(* CODESYS project MID_RunTime_Demo.project

Project tree, tasks and I/O mapping:
  Device : Changsha Xiangji-ARM Cortex A9(xilinx zynq7000)-linux, Changsha Xiangji Hiden Technology Co.Ltd, version 3.5.10.20
    application Application
      libraries: Standard, * (System); SysFile, * (System); SysTypes2 Interfaces, * (System)
      task MainTask (cyclic, interval 4 ms, priority 1) calls PLC_PRG
      task VISU_TASK (cyclic, interval 100 ms, priority 31) calls VisuElems.Visu_Prg
      program PLC_PRG [ST]
      function fn_set_Run_min [ST]
      function read_run_min [ST]
      visualisation RunTime_Visua
      global variables GVL
    SoftMotion General Axis Pool
  text list GlobalTextList
*)

// Device/Application/GVL
{attribute 'qualified_only'}
{attribute 'qualified_only'}


VAR_GLOBAL


	read_runmin:BOOL;
	boot_flag:BOOL;

END_VAR

// Device/Application/PLC_PRG
PROGRAM PLC_PRG
VAR
	Work_min:INT;
	Work_mins:STRING;
	Work_hour:REAL;
	ton1:TON;
	ton2:TON;
	
	new_Run_min:STRING;
	Run_min:STRING;
END_VAR

IF  gvl.boot_flag=FALSE THEN           //上电读一次小时计
   read_run_min(ADR(Work_mins));  //读小时计
   Work_min:=STRING_TO_INT(Work_mins);
   Work_hour:=ANY_TO_REAL(Work_min)/60;
    gvl.boot_flag:=TRUE;
END_IF



//更新小时计
	TON1(IN:=TRUE,PT:=T#60S);
		IF TON1.Q=TRUE THEN
				Work_min:=Work_min+1;		//每分钟加1
				new_Run_min:=INT_TO_STRING(Work_min);
                IF fn_set_Run_min(ADR(new_Run_min), len(new_Run_min)) THEN  //每分钟更新小时计后写入文件
	               Run_min := new_Run_min;
                END_IF				
				
			  TON1(IN:=FALSE,PT:=T#60S);
		END_IF
//读小时计（每6分钟即0.1h读一次）
	TON2(IN:=TRUE,PT:=T#360S);
		IF TON2.Q=TRUE THEN
	          read_run_min(ADR(Work_mins));  //读小时计
              Work_min:=STRING_TO_INT(Work_mins);
              Work_hour:=ANY_TO_REAL(Work_min)/60;	
			  TON2(IN:=FALSE,PT:=T#360S);
		END_IF

END_PROGRAM

// Device/Application/read_run_min
FUNCTION read_run_min : LINT
VAR_INPUT
	runmin: POINTER TO LINT;
END_VAR
VAR
	hFile: RTS_IEC_HANDLE;
	udiOpenError: RTS_IEC_RESULT;
	udiReadError: RTS_IEC_RESULT;
	i :INT;
	iTemp: UDINT;
	udiPos: UDINT;
	str_size: __XWORD;
	udiByteRead: LWORD;

	len_of_line: INT;
	len_of_number :INT;
	magicNumber:REAL;
	check_sum:REAL:= 0;
	temp_num:REAL;
END_VAR

gvl.read_runmin := FALSE;

//检测文件是否存在
hFile := sysfileopen(szFile := '/userapp/r_mins.txt', am := sysfile.AM_READ, pResult:= ADR(udiOpenError));
IF hFile = RTS_INVALID_HANDLE	THEN  //文件不存在
	RETURN;
END_IF
//文件存在，开始读取内容
udiPos := SysFileSetPos(hFile:=hFile, ulOffset := 0);
udiByteRead := sysfile.SysFileRead(hfile := hFile,pbyBuffer := runmin, ulSize := 32, pResult := ADR(udiReadError));
IF udiByteRead < 4 THEN  //读取失败
	sysfile.SysFileClose(hFile := hFile);
	RETURN;
END_IF

gvl.read_runmin := TRUE;

END_FUNCTION

// Device/Application/fn_set_Run_min
FUNCTION fn_set_Run_min : BOOL
VAR_INPUT
	Run_min: POINTER TO STRING;
	len:DINT;
END_VAR
VAR
	hFile: RTS_IEC_HANDLE;
	udiOpenError: RTS_IEC_RESULT;
	udiReadError: RTS_IEC_RESULT;
	udiWriteError: RTS_IEC_RESULT;
	i :INT;
	iTemp: UDINT;
	udiPos: UDINT;
	str_size: __XWORD;
	udiByteRead: UDINT;

	len_of_line: INT;
	len_of_number :INT;
	magicNumber:REAL;
	check_sum:REAL:= 0;
	temp_num:REAL;
	udiByteWrite: LWORD;
END_VAR


fn_set_Run_min := FALSE;

hFile := sysfileopen(szFile := '/userapp/r_mins.txt', am := sysfile.AM_WRITE, pResult := ADR(udiOpenError));
IF hFile = RTS_INVALID_HANDLE THEN //创建文件失败
	RETURN;
END_IF

udiPos := SysFileSetPos(hFile:=hFile, ulOffset:=0);	
udiByteWrite := sysfile.SysFileWrite(hFile := hFile,pbyBuffer := Run_min,ulSize := ANY_TO_DWORD(len), pResult := ADR(udiWriteError));
IF udiByteWrite = 0 THEN
	RETURN;
END_IF

fn_set_Run_min := TRUE;
RETURN;

END_FUNCTION

// Device/Application/RunTime_Visua
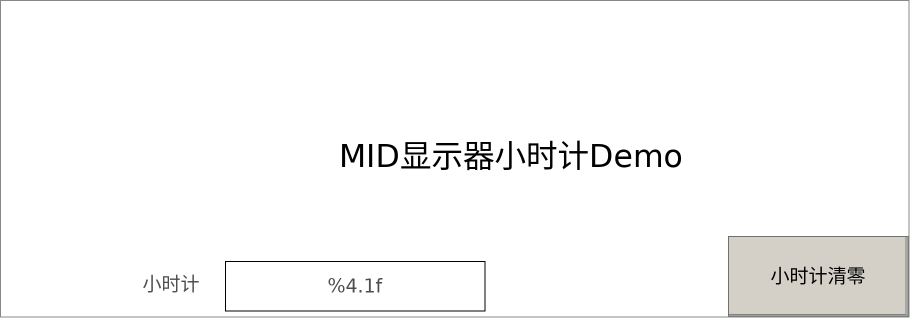
VISUALIZATION RunTime_Visua  // 910x318
    Button (728,236 180x80), "小时计清零"
        OnMouseClick: execute {
            PLC_PRG.new_Run_min:='0';
            IF fn_set_Run_min(ADR(PLC_PRG.new_Run_min), len(PLC_PRG.new_Run_min)) THEN  //每分钟更新小时计后写入文件
            	PLC_PRG.Run_min := PLC_PRG.new_Run_min;
            END_IF
        }
    Label (224,113 574x86), "MID显示器小时计Demo"
    Label (65,254 212x60), "小时计"
    Rectangle (225,261 260x50), "%4.1f", text variable: PLC_PRG.Work_hour
END_VISUALIZATION
